RoboDK station: JuanYMateoLab2.rdk

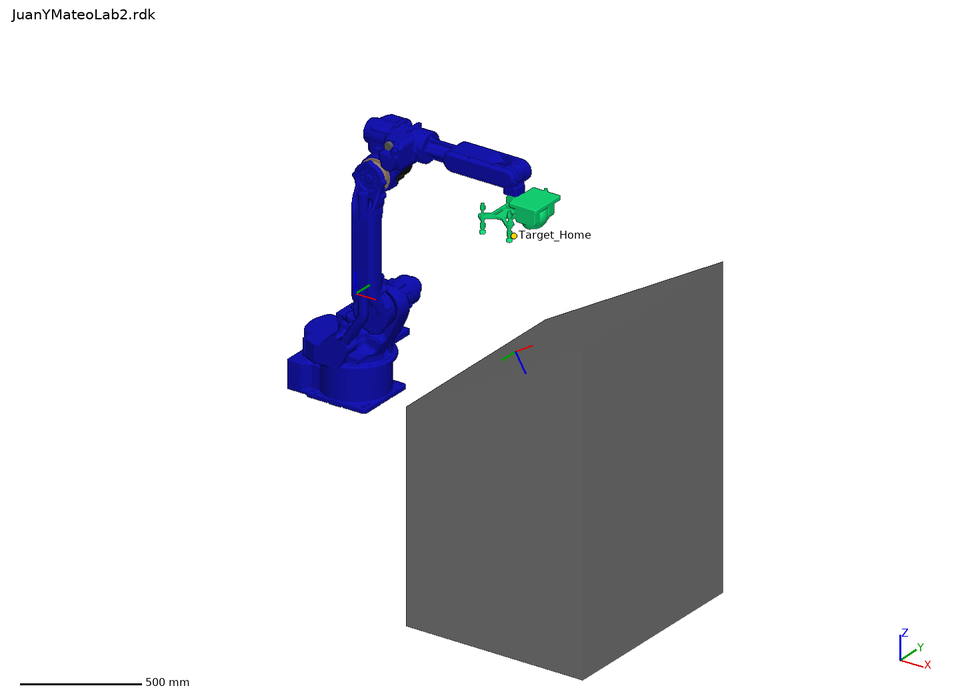
[picture v0: the station drawn from its stored meshes, robots at their saved joint values, targets as dots, program paths as lines]
Station JuanYMateoLab2 (saved by RoboDK 6.0.3). Poses are relative to the parent item; angles as X-Y-Z fixed-axis rotations.
  - frame Motoman MH6 Base at (0, 0, 450) mm
    - robot Motoman MH6: 6 axes, payload 6 kg, reach 1422 mm, repeatability 0.08 mm, weight 130 kg
        modified DH rows (alpha deg, a mm, theta deg, d mm): 0, 0, 0, 450; -90, 152, -90, 0; 0, 614, 0, 0; -90, 155, 0, 640; 90, 0, 90, 0; -90, 0, 0, 95
        base shift (0, 0, -450) mm
        joint limits [-170, -90, -175, -180, -45, -360] to [170, 155, 250, 180, 225, 360]; home [0, 0, 0, 0, 0, 0]; saved at [0, 0, 0, 0, 0, 0]
      - tool Ventosas, TCP at (0, 0, 190) mm, size 250 x 290 x 148 mm
    - frame Frame_from_Target1 at (823.2, -34.49, -21.13) mm, rotated rx -180 ry -30 rz 0 deg
      - target Target_Home (Cartesian target) at (225.55, -34.49, -453.06) mm, rotated rx 0 ry -30 rz 0 deg; joints [0, 0, 0, 0, 0, 0] of Motoman MH6
  - object CAJA2 at (1600, 500, 300) mm, rotated rx 180 ry 0 rz 0 deg, size 886.4 x 1000 x 1511.7 mm, geometry from CAJA2.stp
  - Python program RosPolar (listed below)

--- Python program RosPolar ---
from robodk.robolink import *    # API para comunicarte con RoboDK
from robodk.robomath import *    # Funciones matemáticas
import math
from matplotlib.textpath import TextPath
from matplotlib.path import Path

#------------------------------------------------
# 1) Conexión a RoboDK e inicialización
#------------------------------------------------
RDK = Robolink()

# Elegir un robot (si hay varios, aparece un popup)
robot = RDK.ItemUserPick("Selecciona un robot", ITEM_TYPE_ROBOT)
if not robot.Valid():
    raise Exception("No se ha seleccionado un robot válido.")

# Conectar al robot físico
#if not robot.Connect():
    #raise Exception("No se pudo conectar al robot. Verifica que esté en modo remoto y que la configuración sea correcta.")

# Confirmar conexión
#if not robot.ConnectedState():
   # raise Exception("El robot no está conectado correctamente. Revisa la conexión.")

#print("Robot conectado correctamente.")

#------------------------------------------------
# 2) Cargar el Frame (ya existente) donde quieres dibujar
#    Ajusta el nombre si tu Frame se llama diferente
#------------------------------------------------
frame_name = "Frame_from_Target1"
frame = RDK.Item(frame_name, ITEM_TYPE_FRAME)
if not frame.Valid():
    raise Exception(f'No se encontró el Frame "{frame_name}" en la estación.')

# Asignamos este frame al robot
robot.setPoseFrame(frame)
# Usamos la herramienta activa
robot.setPoseTool(robot.PoseTool())

# Ajustes de velocidad y blending
robot.setSpeed(300)   # mm/s - Ajusta según necesites
robot.setRounding(5)  # blending (radio de curvatura)

#------------------------------------------------
# 3) Parámetros de la figura (rosa polar)
#------------------------------------------------
num_points = 720       # Cuántos puntos muestreamos (mayor = más suave)
A = 70               # Amplitud (Tamaño Del corazon)
z_surface = 0          # Z=0 en el plano del frame
z_safe = -50            # Altura segura para aproximarse y salir

#------------------------------------------------
# 4) Movimiento al centro en altura segura
#------------------------------------------------
# 4) Movimiento a Home

home_target = RDK.Item("Target_Home", ITEM_TYPE_TARGET)
robot.MoveJ(home_target)
# El centro inicio del corazon corresponde a x=500, y=se calcula con el punto inicial del corazon
theta = 0
r = A * ((math.sin(theta) * (math.sqrt(abs(math.cos(theta))) / (math.sin(theta) + 1.4))) - 2 * math.sin(theta) + 2)

robot.MoveJ(transl(500,-r , z_surface + z_safe))

# Bajamos a la "superficie" (Z=0)
robot.MoveL(transl(500, -r, z_surface))

#------------------------------------------------
# 5) Dibujar El Corazon
#    r = A * ((math.sin(theta) * (math.sqrt(abs(math.cos(theta))) / (math.sin(theta) + 1.4))) - 2 * math.sin(theta) + 2)
#    xbase = r * math.cos(theta)
#    ybase = r * math.sin(theta)
#    x = ybase+300
#    y = -xbase
#------------------------------------------------
# Recorremos theta de 0 a 2*pi (una vuelta completa)

full_turn = 2*math.pi


for i in range(num_points+1):
    print(i)
    # Fracción entre 0 y 1
    t = i / num_points
    # Ángulo actual
    theta = full_turn * t

    # Calculamos r
    r = A * ((math.sin(theta) * (math.sqrt(abs(math.cos(theta))) / (math.sin(theta) + 1.4))) - 2 * math.sin(theta) + 2)

    # Convertimos a coordenadas Cartesianas X, Y
    xbase = r * math.cos(theta)
    ybase = r * math.sin(theta)

    x = ybase+500
    y = -xbase

    # Movemos linealmente (MoveL) en el plano del Frame
    robot.MoveL(transl(x, y, z_surface))

# Al terminar, subimos de nuevo para no chocar
robot.MoveL(transl(x, y, z_surface + z_safe))

#Nombres de los integrantes (50) de altura



text = "Juan Andrés"
scale = 1.5             # escalado (para probar tamaños)
letter_spacing = 50       # separación entre letras en X (en el frame del objeto es y positivo)
text_offset_x = -300       # donde empieza el texto en X (en el frame del objeto es y positivo)
text_offset_y = 90 # debajo del corazon en Y (en el frame del objeto es x positivo)

x_cursor = text_offset_x  # cursor que avanza en X por cada letra

for char in text:
    tp = TextPath((0, 0), char, size=50)
    verts = tp.vertices * scale
    codes = tp.codes

    last_x, last_y = None, None

    for (vx, vy), code in zip(verts, codes):
        x_pos = x_cursor + vx
        y_pos = text_offset_y + vy

        if code == Path.MOVETO:
            robot.MoveL(transl(y_pos, x_pos, z_safe))
            robot.MoveL(transl(y_pos, x_pos, z_surface))
        elif code in (Path.LINETO, Path.CURVE3, Path.CURVE4):
            robot.MoveL(transl(y_pos, x_pos, z_surface))

        # Actualiza última posición
        last_x, last_y = x_pos, y_pos

    # Al terminar la letra, solo levanta en el mismo sitio
    if last_x is not None and last_y is not None:
        robot.MoveL(transl(last_y, last_x, z_safe))

    # Avanza cursor para la siguiente letra
    x_cursor += letter_spacing
# Y
text2 = "Y"
x_cursor = -50     # reinicia el cursor horizontal
text_offset_y -= 70  # baja el texto

for char in text2:
    tp = TextPath((0, 0), char, size=50)
    verts = tp.vertices * scale
    codes = tp.codes

    last_x, last_y = None, None

    for (vx, vy), code in zip(verts, codes):
        x_pos = x_cursor + vx
        y_pos = text_offset_y + vy

        if code == Path.MOVETO:
            robot.MoveL(transl(y_pos, x_pos, z_safe))
            robot.MoveL(transl(y_pos, x_pos, z_surface))
        elif code in (Path.LINETO, Path.CURVE3, Path.CURVE4):
            robot.MoveL(transl(y_pos, x_pos, z_surface))

        last_x, last_y = x_pos, y_pos

    # Levantar pluma al terminar la letra
    if last_x is not None and last_y is not None:
        robot.MoveL(transl(last_y, last_x, z_safe))

    # Avanzar cursor para la siguiente letra
    x_cursor += letter_spacing

# segundo nombre
text2 = "Mateo"
x_cursor = -150      # reinicia el cursor horizontal
text_offset_y -= 70  # baja el texto

for char in text2:
    tp = TextPath((0, 0), char, size=50)
    verts = tp.vertices * scale
    codes = tp.codes

    last_x, last_y = None, None

    for (vx, vy), code in zip(verts, codes):
        x_pos = x_cursor + vx
        y_pos = text_offset_y + vy

        if code == Path.MOVETO:
            robot.MoveL(transl(y_pos, x_pos, z_safe))
            robot.MoveL(transl(y_pos, x_pos, z_surface))
        elif code in (Path.LINETO, Path.CURVE3, Path.CURVE4):
            robot.MoveL(transl(y_pos, x_pos, z_surface))

        last_x, last_y = x_pos, y_pos

    # Levantar pluma al terminar la letra
    if last_x is not None and last_y is not None:
        robot.MoveL(transl(last_y, last_x, z_safe))

    # Avanzar cursor para la siguiente letra
    x_cursor += letter_spacing

robot.MoveJ(home_target)

print(f"¡Figura De Corazon completada en el frame '{frame_name}'!")
